TYPE PULSE :
STRUCT
	tLow: TIME   := T#0MS;
	tHigh: TIME := T#0MS;
END_STRUCT
END_TYPE

(* stored: Version 1.1.0.1, ProductVersion 3.1.4024.15
   DUT PULSE: Id {2f52b313-e062-4f00-b14d-0e2773929dff} *)
